{attribute 'GeneratedUsingTerminal: EL3182-0000-0016'}
{attribute addProperty BoxType "EL3182-0000-0016"}
{attribute addProperty Id "StatusAT %I*Status_05CE4FB58ValueAT %I*INT2"}
{attribute addProperty CRC "1200930947"}
{attribute addProperty Size "10"}
TYPE Ch_1_Al_Inputs_4794C083 :
STRUCT
	{attribute addProperty Name "Status"}
	Status AT %I* : Status_05CE4FB5;
	{attribute addProperty Name "Value"}
	Value AT %I* : INT;
END_STRUCT
END_TYPE

(* stored: Version 1.2.0.0, ProductVersion 3.1.4024.9
   DUT Ch_1_Al_Inputs_4794C083: Id {c939f8a5-9030-44ac-9ed7-043312eb4ce3} *)
